Staubli VAL3: clkValve11.pgx

program clkValve11()
begin
  call toggleValve(11)
end
